(* CODESYS project GitDemo

Project tree, tasks and I/O mapping:
  XC204_1 : XC204, Eaton Automation, version 3.5.19.61
      unmapped channels: Output, Input
    application Application
      libraries: Standard, 3.5.18.0 (System); EA_XN300_CAN, 3.5.19.30 (Eaton Automation); EA_XN322_2SI_RS, 3.5.18.2 (Eaton Automation); EA_XN300local_ext, 3.5.19.30 (Eaton Automation)
      task EtherCAT_Task (cyclic, interval t#4ms, priority 1) calls nothing
      task MainTask (cyclic, interval t#10ms, priority 1) calls PLC_PRG, XN300Local
      program PLC_PRG [ST]
      program XN300Local [ST]
    EtherCAT_Master : EtherCAT Master, CODESYS, version 4.8.0.0
        settings: SlaveAutoRestart = True; NetworkName = 'eth1'; NetworkName = "eth1"; SrcAddress1 = 5; SrcAddress2 = 1258783711
      XN_312_GW_EC_1 : XN-312-GW-EC (Eaton SDIAS XN-312-GW-EtherCAT Gateway), Eaton Industries GmbH, order no. XN-312-GW-EC, version Revision=16#00000000
          settings: StationAlias = 0; DC sync0 cycletime = 4000; DC sync1 cycletime = 4000
    XN300_Master : XN300-Master, Eaton Automation, version 3.5.10.0
      XN_322_20DI_PD : XN-322-20DI-PD, Eaton Automation, order no. 8001, version 3.5.10.0
          unmapped channels: Inputs
      XN_322_2DMS_WM_1 : XN-322-2DMS-WM, Eaton Automation, order no. 8006, version 3.5.10.0
          unmapped channels: InputChannel1, InputChannel2, ADC1Diag, ADC2Diag, ModuleDiag
      XN_322_8AIO_I_1 : XN-322-8AIO-I, Eaton Automation, order no. 8012, version 3.5.20.0
          unmapped channels: OutputChannel1, OutputChannel2, OutputChannel3, OutputChannel4, InputChannel1, InputChannel2, InputChannel3, InputChannel4, ModuleDiag, WireBreakDiag
  XC204 : XC204, Eaton Automation, version 3.5.19.61
      unmapped channels: Output, Input
    application Application
      libraries: EA_XN300_CAN, 3.5.19.30 (Eaton Automation); Standard, 3.5.18.0 (System); CAA CiA 405, 4.1.0.0 (CAA Technical Workgroup); MemoryUtils, * (3S - Smart Software Solutions GmbH); StringUtils, 3.5.18.0 (System)
      task MainTask (cyclic, interval t#10ms, priority 1) calls CANopenEnDisableDeviceExample, CANopenManagerExamples, CANbusExamples
      CANbus Examples/
        program CANbusExamples [ST]
        Change CANbus settings (Reconfigure)/
          program ChangeBaudrate [ST]
          program EnableDisableCANbus [ST]
        Query CANbus/
          function GetCANbus [ST]
      CANopen Master Examples/
        program CANopenManagerExamples [ST]
        CiA405/
          Diagnosis/
            EMCY/
              program ReceiveEMCYFromAllDevicesExample [ST]
              program ReceiveEMCYFromOneDeviceExample [ST]
            State/
              program GetCANopenKernelStateExample [ST]
              program GetStateExample [ST]
          Network management/
            program GetCANopenManagerNodeIDExample [ST]
            program NMT_Example [ST]
          SDO access/
            Block and Segmented/
              program SegmentedAndBlockReadExample [ST]
              program SegmentedAndBlockWriteExample [ST]
            Expedited (<= 4byte)/
              program ExpeditedReadExample [ST]
              program ExpeditedWriteExample [ST]
        Stack API/
          program CANopenManagerAPI [ST]
          program CANopenRemoteDeviceAPI [ST]
          Events/
            function block CANopenManagerEventHandler [ST]: EventCallback
      program CANopenEnDisableDeviceExample [ST]
    CANbus : CANbus, Eaton Automation, version 4.2.0.0
      CANopen_Manager : CANopen_Manager, Eaton Automation, version 4.2.0.0
          settings: ConfigVersion = 50659584
        XN_312_GW_CAN : XN-312-GW-CAN, Eaton Automation, order no. 178782, version Revision=16#00000000, FileVersion=1.12
            settings: NODEIDSAVED = 2; SDO Timeout = 1000000; PDO_Autoconfig = TRUE; EXPERTSETTINGS = True; Nodeguarding.Guard Time = 0 ms; Nodeguarding.Life Time Factor = 0; Emergency-General Parameters.Emergency COBID = 16#00000082; Heartbeat-Producer Time = 200; Settings.COBID = 16#00000202; Settings.Transmission Type = 16#FF; Settings.available PDO-Parameter.Inhibit Time available = FALSE; Settings.available PDO-Parameter.Event Timer available = FALSE; Settings.Inhibit Time = 0; Settings.Event Timer = 0; Generic COBID = '$NODEID+16#0200'; Process by CANopenManager = TRUE; Settings.COBID = 16#00000182; Settings.Transmission Type = 16#FF; Settings.available PDO-Parameter.Inhibit Time available = TRUE; Settings.available PDO-Parameter.Event Timer available = TRUE; Settings.Inhibit Time = 0; Settings.Event Timer = 0; Generic COBID = '$NODEID+16#0180'; Process by CANopenManager = TRUE; Settings.COBID = 16#00000282; Settings.Transmission Type = 16#FF; Settings.available PDO-Parameter.Inhibit Time available = TRUE; Settings.available PDO-Parameter.Event Timer available = TRUE; Settings.Inhibit Time = 0; Settings.Event Timer = 0; Generic COBID = '$NODEID+16#0280'; Process by CANopenManager = TRUE; Heartbeat-Consuming1.Heartbeat-Time = 300 ms; Q-Byte : XN_322_16MIO_DIOAI.Index = 16#6200; Q-Byte : XN_322_16MIO_DIOAI.Subindex = 16#01; Q-Byte : XN_322_16MIO_DIOAI.ObjectLength = 8; I-Byte : XN_322_16MIO_DIOAI.Index = 16#6000; I-Byte : XN_322_16MIO_DIOAI.Subindex = 16#01; I-Byte : XN_322_16MIO_DIOAI.ObjectLength = 8; I-Byte : XN_322_16MIO_DIOAI.Index = 16#6000;
              I-Byte : XN_322_16MIO_DIOAI.Subindex = 16#02; I-Byte : XN_322_16MIO_DIOAI.ObjectLength = 8; I-Byte : XN_322_20DI_PCNT.Index = 16#6000; I-Byte : XN_322_20DI_PCNT.Subindex = 16#03; I-Byte : XN_322_20DI_PCNT.ObjectLength = 8; I-Byte : XN_322_20DI_PCNT.Index = 16#6000; I-Byte : XN_322_20DI_PCNT.Subindex = 16#04; I-Byte : XN_322_20DI_PCNT.ObjectLength = 8; I-Byte : XN_322_20DI_PCNT.Index = 16#6000; I-Byte : XN_322_20DI_PCNT.Subindex = 16#05; I-Byte : XN_322_20DI_PCNT.ObjectLength = 8; I-WORD : XN_322_16MIO_DIOAI.Index = 16#6401; I-WORD : XN_322_16MIO_DIOAI.Subindex = 16#01; I-WORD : XN_322_16MIO_DIOAI.ObjectLength = 16; I-WORD : XN_322_16MIO_DIOAI.Index = 16#6401; I-WORD : XN_322_16MIO_DIOAI.Subindex = 16#02; I-WORD : XN_322_16MIO_DIOAI.ObjectLength = 16; SDO List.Set COB-ID sync.Index = 16#1005; SDO List.Set COB-ID sync.Subindex = 16#00; SDO List.Set COB-ID sync.Value = 16#00000080; SDO List.Set COB-ID sync.Size = 32; SDO List.Set COB-ID sync.AbortIfError = FALSE; SDO List.Set COB-ID sync.JumpToLine = FALSE; SDO List.Set COB-ID sync.Line = 0; SDO List.Set Guardtime.Index = 16#100C; SDO List.Set Guardtime.Subindex = 16#00; SDO List.Set Guardtime.Value = 16#00000000; SDO List.Set Guardtime.Size = 16; SDO List.Set Guardtime.AbortIfError = FALSE; SDO List.Set Guardtime.JumpToLine = FALSE; SDO List.Set Guardtime.Line = 0; SDO List.Set Lifetime.Index = 16#100D; SDO List.Set Lifetime.Subindex = 16#00; SDO List.Set Lifetime.Value = 16#00000000; SDO List.Set Lifetime.Size = 8; SDO List.Set Lifetime.AbortIfError = FALSE; SDO List.Set Lifetime.JumpToLine = FALSE; SDO List.Set Lifetime.Line = 0; SDO List.Disable Emcy CobID.Index = 16#1014; SDO List.Disable Emcy CobID.Subindex = 16#00;
              SDO List.Disable Emcy CobID.Value = 16#80000082; SDO List.Disable Emcy CobID.Size = 32; SDO List.Disable Emcy CobID.AbortIfError = FALSE; SDO List.Disable Emcy CobID.JumpToLine = FALSE; SDO List.Disable Emcy CobID.Line = 0; SDO List.Set Emcy CobID.Index = 16#1014; SDO List.Set Emcy CobID.Subindex = 16#00; SDO List.Set Emcy CobID.Value = 16#00000082; SDO List.Set Emcy CobID.Size = 32; SDO List.Set Emcy CobID.AbortIfError = FALSE; SDO List.Set Emcy CobID.JumpToLine = FALSE; SDO List.Set Emcy CobID.Line = 0; SDO List.Set Heartbeat Consumer.Index = 16#1016; SDO List.Set Heartbeat Consumer.Subindex = 16#01; SDO List.Set Heartbeat Consumer.Value = 16#0001012C; SDO List.Set Heartbeat Consumer.Size = 32; SDO List.Set Heartbeat Consumer.AbortIfError = FALSE; SDO List.Set Heartbeat Consumer.JumpToLine = FALSE; SDO List.Set Heartbeat Consumer.Line = 0; SDO List.Set Heartbeat Consumer.Index = 16#1016; SDO List.Set Heartbeat Consumer.Subindex = 16#02; SDO List.Set Heartbeat Consumer.Value = 0; SDO List.Set Heartbeat Consumer.Size = 32; SDO List.Set Heartbeat Consumer.AbortIfError = FALSE; SDO List.Set Heartbeat Consumer.JumpToLine = FALSE; SDO List.Set Heartbeat Consumer.Line = 0; SDO List.Set Heartbeat Consumer.Index = 16#1016; SDO List.Set Heartbeat Consumer.Subindex = 16#03; SDO List.Set Heartbeat Consumer.Value = 0; SDO List.Set Heartbeat Consumer.Size = 32; SDO List.Set Heartbeat Consumer.AbortIfError = FALSE; SDO List.Set Heartbeat Consumer.JumpToLine = FALSE; SDO List.Set Heartbeat Consumer.Line = 0; SDO List.Set Heartbeat Consumer.Index = 16#1016; SDO List.Set Heartbeat Consumer.Subindex = 16#04; SDO List.Set Heartbeat Consumer.Value = 0; SDO List.Set Heartbeat Consumer.Size = 32; SDO List.Set Heartbeat Consumer.AbortIfError = FALSE; SDO List.Set Heartbeat Consumer.JumpToLine = FALSE; SDO List.Set Heartbeat Consumer.Line = 0;
              SDO List.Set Heartbeat Producer.Index = 16#1017; SDO List.Set Heartbeat Producer.Subindex = 16#00; SDO List.Set Heartbeat Producer.Value = 16#000000C8; SDO List.Set Heartbeat Producer.Size = 16; SDO List.Set Heartbeat Producer.AbortIfError = FALSE; SDO List.Set Heartbeat Producer.JumpToLine = FALSE; SDO List.Set Heartbeat Producer.Line = 0; SDO List.Disable PDO.Index = 16#1400; SDO List.Disable PDO.Subindex = 16#01; SDO List.Disable PDO.Value = 16#80000202; SDO List.Disable PDO.Size = 32; SDO List.Disable PDO.AbortIfError = FALSE; SDO List.Disable PDO.JumpToLine = FALSE; SDO List.Disable PDO.Line = 0; SDO List.Set transmission type.Index = 16#1400; SDO List.Set transmission type.Subindex = 16#02; SDO List.Set transmission type.Value = 16#FF; SDO List.Set transmission type.Size = 8; SDO List.Set transmission type.AbortIfError = FALSE; SDO List.Set transmission type.JumpToLine = FALSE; SDO List.Set transmission type.Line = 0; SDO List.Clear pdo mapping.Index = 16#1600; SDO List.Clear pdo mapping.Subindex = 16#00; SDO List.Clear pdo mapping.Value = 16#0; SDO List.Clear pdo mapping.Size = 8; SDO List.Clear pdo mapping.AbortIfError = FALSE; SDO List.Clear pdo mapping.JumpToLine = FALSE; SDO List.Clear pdo mapping.Line = 0; SDO List.Set Mapping.Index = 16#1600; SDO List.Set Mapping.Subindex = 16#01; SDO List.Set Mapping.Value = 16#62000108; SDO List.Set Mapping.Size = 32; SDO List.Set Mapping.AbortIfError = FALSE; SDO List.Set Mapping.JumpToLine = FALSE; SDO List.Set Mapping.Line = 0; SDO List.Set number of mappings.Index = 16#1600; SDO List.Set number of mappings.Subindex = 16#00; SDO List.Set number of mappings.Value = 16#01; SDO List.Set number of mappings.Size = 8; SDO List.Set number of mappings.AbortIfError = FALSE;
              SDO List.Set number of mappings.JumpToLine = FALSE; SDO List.Set number of mappings.Line = 0; SDO List.Set and enable COB-ID.Index = 16#1400; SDO List.Set and enable COB-ID.Subindex = 16#01; SDO List.Set and enable COB-ID.Value = 16#00000202; SDO List.Set and enable COB-ID.Size = 32; SDO List.Set and enable COB-ID.AbortIfError = FALSE; SDO List.Set and enable COB-ID.JumpToLine = FALSE; SDO List.Set and enable COB-ID.Line = 0; SDO List.Disable PDO.Index = 16#1800; SDO List.Disable PDO.Subindex = 16#01; SDO List.Disable PDO.Value = 16#80000182; SDO List.Disable PDO.Size = 32; SDO List.Disable PDO.AbortIfError = FALSE; SDO List.Disable PDO.JumpToLine = FALSE; SDO List.Disable PDO.Line = 0; SDO List.Set transmission type.Index = 16#1800; SDO List.Set transmission type.Subindex = 16#02; SDO List.Set transmission type.Value = 16#FF; SDO List.Set transmission type.Size = 8; SDO List.Set transmission type.AbortIfError = FALSE; SDO List.Set transmission type.JumpToLine = FALSE; SDO List.Set transmission type.Line = 0; SDO List.Set inhibit time.Index = 16#1800; SDO List.Set inhibit time.Subindex = 16#03; SDO List.Set inhibit time.Value = 16#0000; SDO List.Set inhibit time.Size = 16; SDO List.Set inhibit time.AbortIfError = FALSE; SDO List.Set inhibit time.JumpToLine = FALSE; SDO List.Set inhibit time.Line = 0; SDO List.Set event time.Index = 16#1800; SDO List.Set event time.Subindex = 16#05; SDO List.Set event time.Value = 16#0000; SDO List.Set event time.Size = 16; SDO List.Set event time.AbortIfError = FALSE; SDO List.Set event time.JumpToLine = FALSE; SDO List.Set event time.Line = 0; SDO List.Clear pdo mapping.Index = 16#1A00; SDO List.Clear pdo mapping.Subindex = 16#00; SDO List.Clear pdo mapping.Value = 16#0;
              SDO List.Clear pdo mapping.Size = 8; SDO List.Clear pdo mapping.AbortIfError = FALSE; SDO List.Clear pdo mapping.JumpToLine = FALSE; SDO List.Clear pdo mapping.Line = 0; SDO List.Set Mapping.Index = 16#1A00; SDO List.Set Mapping.Subindex = 16#01; SDO List.Set Mapping.Value = 16#60000108; SDO List.Set Mapping.Size = 32; SDO List.Set Mapping.AbortIfError = FALSE; SDO List.Set Mapping.JumpToLine = FALSE; SDO List.Set Mapping.Line = 0; SDO List.Set Mapping.Index = 16#1A00; SDO List.Set Mapping.Subindex = 16#02; SDO List.Set Mapping.Value = 16#60000208; SDO List.Set Mapping.Size = 32; SDO List.Set Mapping.AbortIfError = FALSE; SDO List.Set Mapping.JumpToLine = FALSE; SDO List.Set Mapping.Line = 0; SDO List.Set Mapping.Index = 16#1A00; SDO List.Set Mapping.Subindex = 16#03; SDO List.Set Mapping.Value = 16#60000308; SDO List.Set Mapping.Size = 32; SDO List.Set Mapping.AbortIfError = FALSE; SDO List.Set Mapping.JumpToLine = FALSE; SDO List.Set Mapping.Line = 0; SDO List.Set Mapping.Index = 16#1A00; SDO List.Set Mapping.Subindex = 16#04; SDO List.Set Mapping.Value = 16#60000408; SDO List.Set Mapping.Size = 32; SDO List.Set Mapping.AbortIfError = FALSE; SDO List.Set Mapping.JumpToLine = FALSE; SDO List.Set Mapping.Line = 0; SDO List.Set Mapping.Index = 16#1A00; SDO List.Set Mapping.Subindex = 16#05; SDO List.Set Mapping.Value = 16#60000508; SDO List.Set Mapping.Size = 32; SDO List.Set Mapping.AbortIfError = FALSE; SDO List.Set Mapping.JumpToLine = FALSE; SDO List.Set Mapping.Line = 0; SDO List.Set number of mappings.Index = 16#1A00;
              SDO List.Set number of mappings.Subindex = 16#00; SDO List.Set number of mappings.Value = 16#05; SDO List.Set number of mappings.Size = 8; SDO List.Set number of mappings.AbortIfError = FALSE; SDO List.Set number of mappings.JumpToLine = FALSE; SDO List.Set number of mappings.Line = 0; SDO List.Set and enable COB-ID.Index = 16#1800; SDO List.Set and enable COB-ID.Subindex = 16#01; SDO List.Set and enable COB-ID.Value = 16#00000182; SDO List.Set and enable COB-ID.Size = 32; SDO List.Set and enable COB-ID.AbortIfError = FALSE; SDO List.Set and enable COB-ID.JumpToLine = FALSE; SDO List.Set and enable COB-ID.Line = 0; SDO List.Disable PDO.Index = 16#1801; SDO List.Disable PDO.Subindex = 16#01; SDO List.Disable PDO.Value = 16#80000282; SDO List.Disable PDO.Size = 32; SDO List.Disable PDO.AbortIfError = FALSE; SDO List.Disable PDO.JumpToLine = FALSE; SDO List.Disable PDO.Line = 0; SDO List.Set transmission type.Index = 16#1801; SDO List.Set transmission type.Subindex = 16#02; SDO List.Set transmission type.Value = 16#FF; SDO List.Set transmission type.Size = 8; SDO List.Set transmission type.AbortIfError = FALSE; SDO List.Set transmission type.JumpToLine = FALSE; SDO List.Set transmission type.Line = 0; SDO List.Set inhibit time.Index = 16#1801; SDO List.Set inhibit time.Subindex = 16#03; SDO List.Set inhibit time.Value = 16#0000; SDO List.Set inhibit time.Size = 16; SDO List.Set inhibit time.AbortIfError = FALSE; SDO List.Set inhibit time.JumpToLine = FALSE; SDO List.Set inhibit time.Line = 0; SDO List.Set event time.Index = 16#1801; SDO List.Set event time.Subindex = 16#05; SDO List.Set event time.Value = 16#0000; SDO List.Set event time.Size = 16; SDO List.Set event time.AbortIfError = FALSE; SDO List.Set event time.JumpToLine = FALSE;
              SDO List.Set event time.Line = 0; SDO List.Clear pdo mapping.Index = 16#1A01; SDO List.Clear pdo mapping.Subindex = 16#00; SDO List.Clear pdo mapping.Value = 16#0; SDO List.Clear pdo mapping.Size = 8; SDO List.Clear pdo mapping.AbortIfError = FALSE; SDO List.Clear pdo mapping.JumpToLine = FALSE; SDO List.Clear pdo mapping.Line = 0; SDO List.Set Mapping.Index = 16#1A01; SDO List.Set Mapping.Subindex = 16#01; SDO List.Set Mapping.Value = 16#64010110; SDO List.Set Mapping.Size = 32; SDO List.Set Mapping.AbortIfError = FALSE; SDO List.Set Mapping.JumpToLine = FALSE; SDO List.Set Mapping.Line = 0; SDO List.Set Mapping.Index = 16#1A01; SDO List.Set Mapping.Subindex = 16#02; SDO List.Set Mapping.Value = 16#64010210; SDO List.Set Mapping.Size = 32; SDO List.Set Mapping.AbortIfError = FALSE; SDO List.Set Mapping.JumpToLine = FALSE; SDO List.Set Mapping.Line = 0; SDO List.Set number of mappings.Index = 16#1A01; SDO List.Set number of mappings.Subindex = 16#00; SDO List.Set number of mappings.Value = 16#02; SDO List.Set number of mappings.Size = 8; SDO List.Set number of mappings.AbortIfError = FALSE; SDO List.Set number of mappings.JumpToLine = FALSE; SDO List.Set number of mappings.Line = 0; SDO List.Set and enable COB-ID.Index = 16#1801; SDO List.Set and enable COB-ID.Subindex = 16#01; SDO List.Set and enable COB-ID.Value = 16#00000282; SDO List.Set and enable COB-ID.Size = 32; SDO List.Set and enable COB-ID.AbortIfError = FALSE; SDO List.Set and enable COB-ID.JumpToLine = FALSE; SDO List.Set and enable COB-ID.Line = 0; ConfigVersion = 50659584
          XN_322_16MIO_DIOAI : XN-322-16MIO-DIOAI, Eaton Automation, order no. 0, version Revision=16#00000000, FileVersion=1.12
              settings: Number of Params = 1; Q-Byte : XN_322_16MIO_DIOAI.Index = 16#6200; Q-Byte : XN_322_16MIO_DIOAI.Subindex = 16#01; Q-Byte : XN_322_16MIO_DIOAI.Startbit = 0; Q-Byte : XN_322_16MIO_DIOAI.Endbit = 7; Number of Params = 4; I-Byte : XN_322_16MIO_DIOAI.Index = 16#6000; I-Byte : XN_322_16MIO_DIOAI.Subindex = 16#01; I-Byte : XN_322_16MIO_DIOAI.Startbit = 0; I-Byte : XN_322_16MIO_DIOAI.Endbit = 7; I-Byte : XN_322_16MIO_DIOAI.Index = 16#6000; I-Byte : XN_322_16MIO_DIOAI.Subindex = 16#02; I-Byte : XN_322_16MIO_DIOAI.Startbit = 0; I-Byte : XN_322_16MIO_DIOAI.Endbit = 7; I-WORD : XN_322_16MIO_DIOAI.Index = 16#6401; I-WORD : XN_322_16MIO_DIOAI.Subindex = 16#01; I-WORD : XN_322_16MIO_DIOAI.Startbit = 0; I-WORD : XN_322_16MIO_DIOAI.Endbit = 15; I-WORD : XN_322_16MIO_DIOAI.Index = 16#6401; I-WORD : XN_322_16MIO_DIOAI.Subindex = 16#02; I-WORD : XN_322_16MIO_DIOAI.Startbit = 0; I-WORD : XN_322_16MIO_DIOAI.Endbit = 15
              unmapped channels: Q-Byte : XN_322_16MIO_DIOAI, I-Byte : XN_322_16MIO_DIOAI, I-Byte : XN_322_16MIO_DIOAI, I-WORD : XN_322_16MIO_DIOAI, I-WORD : XN_322_16MIO_DIOAI
          XN_322_20DI_PCNT : XN-322-20DI-PCNT, Eaton Automation, order no. 0, version Revision=16#00000000, FileVersion=1.12
              settings: Number of Params = 3; I-Byte : XN_322_20DI_PCNT.Index = 16#6000; I-Byte : XN_322_20DI_PCNT.Subindex = 16#03; I-Byte : XN_322_20DI_PCNT.Startbit = 0; I-Byte : XN_322_20DI_PCNT.Endbit = 7; I-Byte : XN_322_20DI_PCNT.Index = 16#6000; I-Byte : XN_322_20DI_PCNT.Subindex = 16#04; I-Byte : XN_322_20DI_PCNT.Startbit = 0; I-Byte : XN_322_20DI_PCNT.Endbit = 7; I-Byte : XN_322_20DI_PCNT.Index = 16#6000; I-Byte : XN_322_20DI_PCNT.Subindex = 16#05; I-Byte : XN_322_20DI_PCNT.Startbit = 0; I-Byte : XN_322_20DI_PCNT.Endbit = 7
              unmapped channels: I-Byte : XN_322_20DI_PCNT, I-Byte : XN_322_20DI_PCNT, I-Byte : XN_322_20DI_PCNT
          XN_322_2SI_RS : XN-322-2SI-RS, Eaton Automation, order no. 0, version Revision=16#00000000, FileVersion=1.12
  text list GlobalTextList
*)

// XC204_1/Application/PLC_PRG
PROGRAM PLC_PRG
VAR
    iState 		: INT := 0;
    reconfig 	: DED.Reconfigure;
	xDisable	: BOOL;
	xEnable	: BOOL;
	fbTRIG_Disable: R_TRIG;
	fbTRIG_Enable: R_TRIG;
	xError: BOOL;
	xDone: BOOL;
END_VAR

fbTRIG_Disable(CLK:= xDisable, Q=> );
fbTRIG_Enable(CLK:= xEnable , Q=> );

(*
CASE iState OF
	
	0: //Enable/Disable slave device: Slave1 (= name in device tree) 
		IF fbTRIG_Enable.Q THEN
			XN_312_GW_CAN.Enable := TRUE;
			XN300_Master.Enable := TRUE;
			xError := FALSE;
			iState := 1;
		ELSIF fbTRIG_Disable.Q THEN
			XN_312_GW_CAN.Enable := FALSE;
			XN300_Master.Enable := FALSE;
			xError := FALSE;
			iState := 1;
		END_IF

    1: //start reconfiguring of fieldbus master
      reconfig(xExecute := TRUE, itfNode := CANopen_Manager);
       IF reconfig.xDone THEN
           iState := 3;
       ELSIF reconfig.xError THEN
           iState := 2;
       END_IF

    2: //reconfiguring error
       //TODO: Add code here
       reconfig(xExecute := FALSE);	
	   xError := TRUE;
	   iState := 0;

    3: //reconfiguring successful ==> slave disabled
       //TODO: Add code here
       reconfig(xExecute := FALSE);
	   xDone := TRUE;
	   iState := 0;

END_CASE

*)

END_PROGRAM

// XC204_1/Application/XN300Local
PROGRAM XN300Local
VAR
	eMasterStatusInfo1: ENUM_MASTERSTATUSINFO;
	sMasterStatusInfo2: STRING;
	uiPeriode: UINT;
	stSlotInfo: EA_XN300local_ext.STRUCT_XNSLOTINFO;
	byData: BYTE;
	xRead: BOOL;
END_VAR

// Get XN300_Master Status
GetXnMasterStatus(peStatusInfo:= ADR(eMasterStatusInfo1), pstrStatusInfo2:= ADR(sMasterStatusInfo2), uiStatusInfo2Length:= LEN(sMasterStatusInfo2));

uiPeriode := GetXnPeriode();

stSlotInfo := GetXnSlotInfo(uiSlotNumber:= 1);

// XN_322_8AO_U2 -> Offset 16#80 -> ModuleDiagnose 1:No power supply, 2:No SyncSignal, 3: FlashCRC Error, 4:RAMCRC Error, 5:FlashMemory Error
IF xRead THEN
	ReadXnDirect(uiModuleNumber:= 1, uiModuleOffset:=16#080 , uiDataLength:= 2, pbyData:= ADR(byData));
	xRead := FALSE;
END_IF

(*
SetXnPeriode(uiXnPeriode:= );

SetXnUserLed(uiModuleNumber:= , uiLedMode:= );

WriteXnDirect(uiModuleNumber:= , uiModuleOffset:= , uiDataLength:= , pbyData:= );
*)

END_PROGRAM

// XC204/Application/CANopenEnDisableDeviceExample
PROGRAM CANopenEnDisableDeviceExample
VAR
    iState 		: INT := 0;
    reconfig 	: DED.Reconfigure;
	xDisable	: BOOL;
	xEnable	: BOOL;
	fbTRIG_Disable: R_TRIG;
	fbTRIG_Enable: R_TRIG;
	xError: BOOL;
	xDone: BOOL;
END_VAR

fbTRIG_Disable(CLK:= xDisable, Q=> );
fbTRIG_Enable(CLK:= xEnable , Q=> );


CASE iState OF
	
	0: //Enable/Disable slave device: Slave1 (= name in device tree) 
		IF fbTRIG_Enable.Q THEN
			XN_312_GW_CAN.Enable := TRUE;
			xError := FALSE;
			iState := 1;
		ELSIF fbTRIG_Disable.Q THEN
			XN_312_GW_CAN.Enable := FALSE;
			xError := FALSE;
			iState := 1;
		END_IF

    1: //start reconfiguring of fieldbus master
      reconfig(xExecute := TRUE, itfNode := CANopen_Manager);
       IF reconfig.xDone THEN
           	iState := 3;
			xDisable := FALSE;
			xEnable := FALSE;
       ELSIF reconfig.xError THEN
           iState := 2;
       END_IF

    2: //reconfiguring error
       //TODO: Add code here
       reconfig(xExecute := FALSE);	
	   xError := TRUE;
	   iState := 0;

    3: //reconfiguring successful ==> slave disabled
       //TODO: Add code here
       reconfig(xExecute := FALSE);
	   xDone := TRUE;
	   iState := 0;

END_CASE

END_PROGRAM

// XC204/Application/CANopen Master Examples/CANopenManagerExamples
PROGRAM CANopenManagerExamples
VAR
END_VAR

///////////////////////////////////////// CIA 405 Examples //////////////////////////////////////////////////////

//Diagnosis Examples
GetStateExample(); //How to get the state of a CANopenRemote Device?
GetCANopenKernelStateExample(); //How to get the CANopen stack kernel state?
ReceiveEMCYFromAllDevicesExample(); //How to check if any CANopenRemote Device has a pending Emergency?
ReceiveEMCYFromOneDeviceExample(); //How to check if a specific CANopenRemote Device has a pending Emergency?

//SDO Examples
ExpeditedReadExample(); //How to read up to 4 bytes by SDO?
ExpeditedWriteExample(); //How to write up to 4 bytes by SDO?
SegmentedAndBlockReadExample(); //How to read more than 4 bytes by SDO?
SegmentedAndBlockWriteExample(); //How to write more than 4 bytes by SDO?

NMT_Example(); //How to start/stop/reset CANopenRemote Devices?

GetCANopenManagerNodeIDExample(); //How to read the CANopen Manager NodeID?

///////////////////////////////////////// General Examples //////////////////////////////////////////////////////

CANopenManagerAPI(); //How to use the CANopen Manager API?
CANopenRemoteDeviceAPI(); //How to use the CANopenRemoteDevice API?

END_PROGRAM

// XC204/Application/CANopen Master Examples/CiA405/Diagnosis/State/GetStateExample
// The following program gets the current CANopen state of the CANopenRemoteDevice attached below the CANopen_Manager.
// Set xEnable to TRUE in online mode to get the program working.
PROGRAM GetStateExample
VAR
	xEnable : BOOL; // Set this variable to true to start the example code. Variable will be set to FALSE if GetState finished execution.
	State : CiA405.DEVICE_STATE; // Result: CANopen State
	
	GetState : CIA405.GET_STATE;
END_VAR

IF GetState.CONFIRM = TRUE THEN
	// GetState successful. Output STATE contains result.
	State := GetState.STATE;
	xEnable := FALSE;
ELSIF GetState.ERROR <> CIA405.CANOPEN_KERNEL_ERROR.CANOPEN_KERNEL_NO_ERROR THEN
	// an error occured while processing GetState e.g. wrong NodeID or NetworkID
	xEnable := FALSE;
END_IF

// GetState needs the CAN network and the device NodeID (input DEVICE). 
GetState( 	ENABLE := xEnable,
		  	NETWORK := CANbus.NetId + 1, //CODESYS NetId starts by 0 (the number entered into the CANbus configurator); CiA405 NETWORK by 1; That is the reason why we have to increment it here.
		  	TIMEOUT := 0, // no timeout for GetState needed because it is processed locally.
			DEVICE := XN_312_GW_CAN.NodeID // Note: If you want to get the state of the CANopenManager, you can use the CANopenManager NodeID or NodeID 0.
												 // A CANopenManager goes to OPERATIONAL if all mandatory (= not optional) slaves are operational.
);

END_PROGRAM

// XC204/Application/CANopen Master Examples/CiA405/Diagnosis/State/GetCANopenKernelStateExample
// This program gets the state of the CANopenManager kernel. If kernel has no error everything is working fine.
// See CiA405.CANOPEN_KERNEL_ERROR in library manager for further details.
// Set xEnable to TRUE in online mode to get the program working.
PROGRAM GetCANopenKernelStateExample
VAR
	xEnable : BOOL; // Set this variable to true to start the example code. Variable will be set to FALSE if GetState finished execution.
	xErrorPending : BOOL; //true if a CANopen Kernel error is pending
	State : CiA405.CANOPEN_KERNEL_ERROR; // Result: CANopen Manager kernel state
	
	GetKernelState : CIA405.GET_CANOPEN_KERNEL_STATE;
END_VAR

IF GetKernelState.CONFIRM = TRUE THEN
	// GetKernelState successful. Output STATE contains result.
	State := GetKernelState.STATE;
	xErrorPending := State <> CIA405.CANOPEN_KERNEL_ERROR.CANOPEN_KERNEL_NO_ERROR;
	xEnable := FALSE;
ELSIF GetKernelState.ERROR <> CIA405.CANOPEN_KERNEL_ERROR.CANOPEN_KERNEL_NO_ERROR THEN
	// an error occured while processing GetKernelState e.g. wrong NetworkID
	xEnable := FALSE;
END_IF

GetKernelState( 	ENABLE := xEnable,
		  			NETWORK := CANbus.NetId + 1, //CODESYS NetId starts by 0 (the number entered into the CANbus configurator); CiA405 NETWORK by 1; That is the reason why we have to increment it here.
		  			TIMEOUT := 0 // no timeout for GetKernelState needed because it is processed locally.
);

END_PROGRAM

// XC204/Application/CANopen Master Examples/CiA405/Diagnosis/EMCY/ReceiveEMCYFromAllDevicesExample
// This program checks if any emergency is pending for any device of a given CANopenManager network.
// Set xEnable to TRUE in online mode to get the program working.
PROGRAM ReceiveEMCYFromAllDevicesExample
VAR
	xEnable : BOOL; // Set this variable to true to start the example code. Variable will be set to FALSE if RecvEMCY finished execution.
	xEMCYPending : BOOL; //true if EMCY is pending ==> see EMCY and NodeID for EMCY information
	EMCY : CIA405.EMCY_ERROR; //contains EMCY information
	NodeID : CIA405.DEVICE; //NodeID of EMCY sender
	
	RecvEMCY : CIA405.RECV_EMCY;
END_VAR

IF RecvEMCY.CONFIRM = TRUE THEN
	// RecvEMCY successful.
	IF RecvEMCY.DEVICE <> 0 THEN
		//an EMCY from NodeID RecvEMCY.DEVICE is pending
		xEMCYPending := TRUE;
		EMCY := RecvEMCY.ERRORINFO;
		NodeID := RecvEMCY.DEVICE;
	ELSE
		//all devices are error free
		xEMCYPending := FALSE;
	END_IF

	xEnable := FALSE;
ELSIF RecvEMCY.ERROR <> CIA405.CANOPEN_KERNEL_ERROR.CANOPEN_KERNEL_NO_ERROR THEN
	// an error occured while processing RecvEMCY e.g. wrong NodeID or NetworkID
	xEnable := FALSE;
END_IF

RecvEMCY( 	ENABLE := xEnable,
		  	NETWORK := CANbus.NetId + 1, //CODESYS NetId starts by 0 (the number entered into the CANbus configurator); CiA405 NETWORK by 1; That is the reason why we have to increment it here.
		  	TIMEOUT := 0 // no timeout for RecvEMCY needed because it is processed locally.
);

END_PROGRAM

// XC204/Application/CANopen Master Examples/CiA405/Diagnosis/EMCY/ReceiveEMCYFromOneDeviceExample
// This program checks if any emergency is pending for CANopenRemoteDevice.
// Set xEnable to TRUE in online mode to get the program working.
PROGRAM ReceiveEMCYFromOneDeviceExample
VAR
	xEnable : BOOL; // Set this variable to true to start the example code. Variable will be set to FALSE if RecvEMCYDev finished execution.
	xEMCYPending : BOOL; //true if EMCY is pending ==> see EMCY for EMCY information
	EMCY : CIA405.EMCY_ERROR; //contains EMCY information
	
	RecvEMCYDev : CIA405.RECV_EMCY_DEV;
END_VAR

IF RecvEMCYDev.CONFIRM = TRUE THEN
	// RecvEMCYDev successful
	IF RecvEMCYDev.ERRORINFO.EMCY_ERROR_CODE <> 0 THEN
		//an EMCY is pending ==> see RecvEMCYDev.ERRORINFO for EMCY information
		xEMCYPending := TRUE;
		EMCY := RecvEMCYDev.ERRORINFO;
	ELSE
		//device is error free
		xEMCYPending := FALSE;
	END_IF
	xEnable := FALSE;
ELSIF RecvEMCYDev.ERROR <> CIA405.CANOPEN_KERNEL_ERROR.CANOPEN_KERNEL_NO_ERROR THEN
	// an error occured while processing RecvEMCY e.g. wrong NodeID or NetworkID
	xEnable := FALSE;
END_IF

RecvEMCYDev( 	ENABLE := xEnable,
		  		NETWORK := CANbus.NetId + 1, //CODESYS NetId starts by 0 (the number entered into the CANbus configurator); CiA405 NETWORK by 1; That is the reason why we have to increment it here.
		  		TIMEOUT := 0, // no timeout for RecvEMCYDev needed because it is processed locally.
				DEVICE := XN_312_GW_CAN.NodeID //NodeID to receive EMCY from
);

END_PROGRAM

// XC204/Application/CANopen Master Examples/CiA405/SDO access/Expedited (<= 4byte)/ExpeditedReadExample
// The following program reads the device type of CANopenRemoteDevice and shows how to usde SDORead4 function block.
// Set xEnable to TRUE in online mode to get the program working.
PROGRAM ExpeditedReadExample
VAR
	xEnable       : BOOL; // Set this variable to true to start the example code. Variable will be set to FALSE if Expedited transfer finished execution.
	dwValue : DWORD; //read value
	dwAbortCode : DWORD; //contains abort code in case of error
	
	SDORead4 	  : CIA405.SDO_READ4;
END_VAR

IF SDORead4.CONFIRM THEN
	//value was read without error
	// ==> Copy data from SDO read function block
	MEMUtils.MemCpy(pbyDest := ADR(dwValue), pbySrc := ADR(SDORead4.DATA[1]), dwSize := SIZEOF(dwValue));
	//==> On big endian systems: dwValue has to be swapped to CANopen byte order (= Little Endian).
	MEMUtils.SwapLocalToIntel(pAddress := ADR(dwValue), iSize := TO_INT(SIZEOF(dwValue))); //function only swaps on big endian systems
	xEnable := FALSE;
ELSIF SDORead4.ERROR <> CiA405.CANOPEN_KERNEL_ERROR.CANOPEN_KERNEL_NO_ERROR THEN
	//Error occured
	IF SDORead4.ERROR = CIA405.CANOPEN_KERNEL_ERROR.CANOPEN_KERNEL_OTHER_ERROR THEN
		//output error info contains abort code in little endian format
		MEMUtils.MemCpy(pbyDest := ADR(dwAbortCode), pbySrc := ADR(SDORead4.ERRORINFO), dwSize := SIZEOF(dwAbortCode));
		MEMUtils.SwapLocalToIntel(pAddress := ADR(dwAbortCode), iSize := TO_INT(SIZEOF(dwAbortCode))); //function only swaps on big endian systems	
	END_IF
	xEnable := FALSE;
END_IF

SDORead4(
	NETWORK:= CANbus.NetId + 1, //CODESYS NetId starts by 0 (the number entered into the CANbus configurator); CiA405 NETWORK by 1; That is the reason why we have to increment it here.
	ENABLE:= xEnable,
	TIMEOUT:= 0, //Timeout for SDO read in ms. Here: 0 ==> no timeout
	DEVICE:= XN_312_GW_CAN.NodeID, // NodeID of destination device
	CHANNEL:= 0, //SDO channel which should be used. 0 means auto channeling ==> the next free channel will be used. It depends on the slave which settings are working here but 0 and channel 1 is always working. 
	INDEX:= 16#1000, //object index which should be read
	SUBINDEX:= 0 //object sub index which should be read
);

END_PROGRAM

// XC204/Application/CANopen Master Examples/CiA405/SDO access/Expedited (<= 4byte)/ExpeditedWriteExample
// The following program writes a 32bit value with SDO expedited transfer.
// Set xEnable to TRUE in online mode to get the program working.
PROGRAM ExpeditedWriteExample
VAR
	xEnable       : BOOL; // Set this variable to true to start the example code. Variable will be set to FALSE if Expedited transfer finished execution.
	diValue : DINT := 10; //value which should be written
	dwAbortCode : DWORD; //contains abort code in case of error
	
	SDOWrite4 	  : CiA405.SDO_WRITE4;
	RTrig 		  : Standard.R_TRIG;
END_VAR

RTrig(CLK := xEnable); //detect a rising edge for xEnable

IF RTrig.Q THEN
	// Rising edge for xEnable detected ==> Prepare SDO write function block
	// ==> Copy data to SDO write function block
	MEMUtils.MemCpy(pbyDest := ADR(SDOWrite4.DATA[1]), pbySrc := ADR(diValue), dwSize := SIZEOF(diValue));
	//==> On big endian systems: diValue has to be swapped to CANopen byte order (= Little Endian).
	MEMUtils.SwapLocalToIntel(pAddress := ADR(SDOWrite4.DATA[1]), iSize := TO_INT(SIZEOF(diValue))); //function only swaps on big endian systems
END_IF

IF SDOWrite4.CONFIRM THEN
	//value was written without error
	xEnable := FALSE;
ELSIF SDOWrite4.ERROR <> CiA405.CANOPEN_KERNEL_ERROR.CANOPEN_KERNEL_NO_ERROR THEN
	//Error occured
	IF SDOWrite4.ERROR = CIA405.CANOPEN_KERNEL_ERROR.CANOPEN_KERNEL_OTHER_ERROR THEN
		//output error info contains abort code in little endian format
		MEMUtils.MemCpy(pbyDest := ADR(dwAbortCode), pbySrc := ADR(SDOWrite4.ERRORINFO), dwSize := SIZEOF(dwAbortCode));
		MEMUtils.SwapLocalToIntel(pAddress := ADR(dwAbortCode), iSize := TO_INT(SIZEOF(dwAbortCode))); //function only swaps on big endian systems	
	END_IF
	xEnable := FALSE;
END_IF

SDOWrite4(
	NETWORK:= CANbus.NetId + 1, //CODESYS NetId starts by 0 (the number entered into the CANbus configurator); CiA405 NETWORK by 1; That is the reason why we have to increment it here.
	ENABLE:= xEnable,
	TIMEOUT:= 0, //Timeout for SDO write in ms. Here: 0 ==> no timeout
	DEVICE:= XN_312_GW_CAN.NodeID, // NodeID of destination device
	CHANNEL:= 0, //SDO channel which should be used. 0 means auto channeling ==> the next free channel will be used. It depends on the slave which settings are working here but 0 and channel 1 is always working. 
	INDEX:= 16#6412, //object index which should be written
	SUBINDEX:= 1, //object sub index which should be written
	DATALENGTH:= TO_USINT(SIZEOF(diValue)) //length of data to be written
);

END_PROGRAM

// XC204/Application/CANopen Master Examples/CiA405/SDO access/Block and Segmented/SegmentedAndBlockReadExample
// This program uses CiA405.SDO_READ_DATA for reading more than 4 byte from a slave using segmented or block transfer.
//
// This example code reads object 16#1008sub0 which is the device name.
// CiA405.SDO_READ_DATA is a universal function block which can be also used for expedited transfer (<= 4byte).
// If you never want to read more than 4 byte use the CIA405.SDO_READ4 functionblock instead.
// Set xEnable to TRUE in online mode to get the program working.
PROGRAM SegmentedAndBlockReadExample
VAR
	xEnable       : BOOL; // Set this variable to true to start the example code.
	psData        : POINTER TO STRING(MAX_CHAR - 1) := ADR(aData); // Result: Device Name
	dwAbortCode	  : DWORD; //contains abort code in case of error

	SDORead    	  : CIA405.SDO_READ_DATA;
	RTrig 		  : Standard.R_TRIG;										  
	aData	      : ARRAY[0..MAX_CHAR] OF BYTE;
	udiDataLength : UDINT;
END_VAR
VAR CONSTANT
	MAX_CHAR : INT := 256;
END_VAR

RTrig(CLK := xEnable);

IF RTrig.Q THEN
	// Rising edge for xEnable detected ==> Prepare SDO write function block
	
	// ==> Initialize read buffer with 0 (clear old read results)
	MEMUtils.MemSet(pbyBuffer := ADR(aData[0]), byValue := 0, dwSize := SIZEOF(aData));
	
	// ==> Set udiDataLength to read buffer length.
	// Note: Do not forget setting udiDataLength each time when you start a new SDO read operation. 
	// This is necessary because udiDataLength is a VAR_IN_OUT variable and will be modified by SDORead function block!
	// It contains the number of valid bytes read by the function block.
	udiDataLength := SIZEOF(aData) - 1; //-1 only needed because CANopen strings are not null terminated! So we need one additional byte for the null termination. ==> Not needed for other datatypes!
END_IF

IF SDORead.CONFIRM THEN
	// SDO Read successful. aData contains data (= Device Name); udiDataLength contains number of bytes read (string length without null termination).
	xEnable := FALSE;
ELSIF SDORead.ERROR <> CiA405.CANOPEN_KERNEL_ERROR.CANOPEN_KERNEL_NO_ERROR THEN
	// Error occured
	IF SDORead.ERROR = CIA405.CANOPEN_KERNEL_ERROR.CANOPEN_KERNEL_OTHER_ERROR THEN
		//output error info contains abort code in little endian format
		MEMUtils.MemCpy(pbyDest := ADR(dwAbortCode), pbySrc := ADR(SDORead.ERRORINFO), dwSize := SIZEOF(dwAbortCode));
		MEMUtils.SwapLocalToIntel(pAddress := ADR(dwAbortCode), iSize := TO_INT(SIZEOF(dwAbortCode))); //function only swaps on big endian systems	
	END_IF
	xEnable := FALSE;
END_IF

SDORead(   Enable     := xEnable,
		   Network    := CANbus.NetId + 1, //CODESYS NetId starts by 0 (the number entered into the CANbus configurator); CiA405 NETWORK by 1; That is the reason why we have to increment it here.
           Timeout    := 0, //Timeout for SDO read in ms. Here: 0 ==> no timeout
           Device     := XN_312_GW_CAN.NodeID, // NodeID of destination device
           Channel    := 0, //SDO channel which should be used. 0 means auto channeling ==> the next free channel will be used. It depends on the slave which settings are working here but 0 and channel 1 is always working. 
           Index      := 16#1008, //object index which should be read ==> 16#1008sub0 = Device Name
           SubIndex   := 0, //object sub index which should be read ==> 16#1008sub0 = Device Name
		   MODE		  := CIA405.SDO_MODE.AUTO, //Use SDO mode AUTO ==> Mode will be selected automatically. Use SDO_MODE.BLOCK for forcing Block Transfer.
           Data       := ADR(aData), // Pointer to data buffer where result should be written to.
           DataLength := udiDataLength //VAR_IN: Length of data buffer; VAR_OUT: Length of data written to data buffer.
);

END_PROGRAM

// XC204/Application/CANopen Master Examples/CiA405/SDO access/Block and Segmented/SegmentedAndBlockWriteExample
// This program uses CiA405.SDO_WRITE_DATA for writing more than 4 byte using segmented or block transfer.
//
// This example code writes a string into object 16#3000 of CANopenRemoteDevice.
// CiA405.SDO_WRITE_DATA is a universal function block which can be also used for expedited transfer (<= 4byte).
// If you never want to write more than 4 byte use the CIA405.SDO_WRITE4 functionblock instead.
// In online mode: Set psData to the string which should be written and then set xEnable to TRUE to get the program working.
// Afterwards you can check result in CANopenLocalDeviceExamples.strTestString. The Variable is mapped to object 16#3000 in object dictionary.
PROGRAM SegmentedAndBlockWriteExample
VAR
	xEnable       : BOOL; // Set this variable to true to start the example code.
	psData        : POINTER TO STRING(MAX_CHAR - 1) := ADR(aData); // String to write
	dwAbortCode	  : DWORD; //contains abort code in case of error

	SDOWrite      : CIA405.SDO_WRITE_DATA;							  
	aData	      : ARRAY[0..MAX_CHAR] OF BYTE;
END_VAR
VAR CONSTANT
	MAX_CHAR : INT := 256;
END_VAR

IF SDOWrite.CONFIRM THEN
	// SDO Write successful.
	xEnable := FALSE;
ELSIF SDOWrite.ERROR <> CiA405.CANOPEN_KERNEL_ERROR.CANOPEN_KERNEL_NO_ERROR THEN
	// Error occured
	IF SDOWrite.ERROR = CIA405.CANOPEN_KERNEL_ERROR.CANOPEN_KERNEL_OTHER_ERROR THEN
		//output error info contains abort code in little endian format
		MEMUtils.MemCpy(pbyDest := ADR(dwAbortCode), pbySrc := ADR(SDOWrite.ERRORINFO), dwSize := SIZEOF(dwAbortCode));
		MEMUtils.SwapLocalToIntel(pAddress := ADR(dwAbortCode), iSize := TO_INT(SIZEOF(dwAbortCode))); //function only swaps on big endian systems	
	END_IF
	xEnable := FALSE;
END_IF

SDOWrite(  Enable     := xEnable,
		   Network    := CANbus.NetId + 1, //CODESYS NetId starts by 0 (the number entered into the CANbus configurator); CiA405 NETWORK by 1; That is the reason why we have to increment it here.
           Timeout    := 0, //Timeout for SDO read in ms. Here: 0 ==> no timeout
           Device     := XN_312_GW_CAN.NodeID, // NodeID of destination device
           Channel    := 0, //SDO channel which should be used. 0 means auto channeling ==> the next free channel will be used. It depends on the slave which settings are working here but 0 and channel 1 is always working. 
           Index      := 16#3000, //object index which should be written ==> 16#3000 = simple string object
           SubIndex   := 0, //object sub index which should be written
		   MODE		  := CIA405.SDO_MODE.AUTO, //Use SDO mode AUTO ==> Mode will be selected automatically. Use SDO_MODE.BLOCK for forcing Block Transfer.
           Data       := ADR(aData), // Pointer to data buffer where result should be written to.
           DataLength := TO_UDINT(Stu.StrLenA(ADR(aData[0]))) //Length of data
);

END_PROGRAM

// XC204/Application/CANopen Master Examples/CiA405/Network management/NMT_Example
// The following program sends a NMT command to the CANopenRemoteDevice attached below the CANopen_Manager.
// Set eState to the desired NMT command and xEnable to TRUE in online mode to get the program working.
PROGRAM NMT_Example
VAR
	xEnable : BOOL; // Set this variable to true to start the example code. Variable will be set to FALSE if NMT finished execution.
	eState : CIA405.TRANSITION_STATE := CIA405.TRANSITION_STATE.RESET_NODE; // NMT command which should be sent.
	
	NMT : CIA405.NMT;
END_VAR

IF NMT.CONFIRM = TRUE THEN
	// NMT command successful.
	xEnable := FALSE;
ELSIF NMT.ERROR <> CIA405.CANOPEN_KERNEL_ERROR.CANOPEN_KERNEL_NO_ERROR THEN
	// an error occured while processing NMT e.g. wrong NodeID or NetworkID
	xEnable := FALSE;
END_IF

NMT(	ENABLE := xEnable,
		NETWORK := CANbus.NetId + 1, //CODESYS NetId starts by 0 (the number entered into the CANbus configurator); CiA405 NETWORK by 1; That is the reason why we have to increment it here.
		TIMEOUT := 0, // no timeout for GetState needed because it is processed locally.
		DEVICE := XN_312_GW_CAN.NodeID, // Use 0 if you want to send a NMT all command!
		STATE := eState //the NMT command which should be sent
);

END_PROGRAM

// XC204/Application/CANopen Master Examples/CiA405/Network management/GetCANopenManagerNodeIDExample
// This program reads the NodeID of the local CANopenManager.
// Set xEnable to TRUE in online mode to get the program working.
PROGRAM GetCANopenManagerNodeIDExample
VAR
	xEnable : BOOL; // Set this variable to true to start the example code. Variable will be set to FALSE if GetNodeID finished execution.
	NodeID : CiA405.DEVICE; // Result: CANopen NodeID
	
	GetNodeID : CIA405.GET_LOCAL_NODE_ID;
END_VAR

IF GetNodeID.CONFIRM = TRUE THEN
	// GetNodeID successful. Output device contains CANopenManager NodeID.
	NodeID := GetNodeID.DEVICE;
	xEnable := FALSE;
ELSIF GetNodeID.ERROR <> CIA405.CANOPEN_KERNEL_ERROR.CANOPEN_KERNEL_NO_ERROR THEN
	// an error occured while processing GetState e.g. wrong NodeID or NetworkID
	xEnable := FALSE;
END_IF

GetNodeID( 	ENABLE := xEnable,
		  	NETWORK := CANbus.NetId + 1, //CODESYS NetId starts by 0 (the number entered into the CANbus configurator); CiA405 NETWORK by 1; That is the reason why we have to increment it here.
		  	TIMEOUT := 0 // no timeout for GetNodeID needed because it is processed locally.
);

END_PROGRAM

// XC204/Application/CANopen Master Examples/Stack API/CANopenManagerAPI
// This example program shows how to use the CANopen Manager API.
PROGRAM CANopenManagerAPI
VAR
	pDevice : POINTER TO _3SCOS.CANRemoteDevice;
	kernelState : _3SCOS.CANOPEN_KERNEL_STATE;
	xAllMandatorySlaveBooted : BOOL;
	xAllOptionalSlavesBooted : BOOL;
	wNMTInhibitTime : WORD;
	
	udiNumberOfSlaves : UDINT; //How many slaves are attached below the CANopenManager
	udiNumberOfOperationalSlaves : UDINT; //How many slaves are in OPERATIONAL
	udiTotalConfigurationErrors : UDINT; //How many configuration errors (= SDO aborts) happened in configuration phase?
	udiNumberOfSlavesWithActivatedErrorControl : UDINT; //How many slaves have Error control (= Heartbeat or Nodeguarding) activated?
	
	usiCurrentNodeID : USINT;
	
	xEventHandlerRegistered : BOOL;
	EventHandler : CANopenManagerEventHandler; // CANopenManager event handler instance
END_VAR

//gets the CANopenManager kernel state ==> see also CiA405.GET_CANOPEN_KERNEL_STATE
kernelState := CANopen_Manager.KernelState;

//Are all mandatory slaves found and configured by CANopenManager?
xAllMandatorySlaveBooted := CANopen_Manager.MandatorySlavesBooted;

//Are all optional slaves found and configured by CANopenManager?
xAllOptionalSlavesBooted := CANopen_Manager.OptionalSlavesBooted;

//Gets or sets the NMT Inhibit Time (unit: multiple of 100us).
wNMTInhibitTime := CANopen_Manager.NMTInhibitTime;

//go through all remote devices of CANopen_Manager and collect some statistics
udiNumberOfSlaves := 0;
udiNumberOfOperationalSlaves := 0;
udiTotalConfigurationErrors := 0;
udiNumberOfSlavesWithActivatedErrorControl := 0;

FOR usiCurrentNodeID := 1 TO 127 DO
	pDevice := CANopen_Manager.GetSlaveByNodeID(usiCurrentNodeID);
	IF pDevice <> 0 THEN
		//count slaves
		udiNumberOfSlaves := udiNumberOfSlaves + 1;
		
		//Get the slave state ==> see also CiA405.GET_STATE
		IF pDevice^.CANopenState = _3SCOS.DEVICE_STATE.OPERATIONAL THEN
			udiNumberOfOperationalSlaves := udiNumberOfOperationalSlaves + 1;
		END_IF
		
		//Sum up configuration errors. 
		//NOTE: For getting more detailed information you can add the Compiler Define CANOPEN_DEBUG to the application.
		//Then perform a new download and go to the PLC logger. It contains further information for debugging purpose. 
		udiTotalConfigurationErrors := udiTotalConfigurationErrors + pDevice^.ConfigurationErrors;
		
		//Sum up all slaves with error control activated
		IF pDevice^.ErrorControlActivated THEN
			udiNumberOfSlavesWithActivatedErrorControl := udiNumberOfSlavesWithActivatedErrorControl + 1;
		END_IF
	END_IF
END_FOR

// Register a CANopen Manager event handler: An event handler can be used to add additional code to the stack state machine.
// In this example a SDO Read for CANopenRemoteDevice is performed after SDO configuration phase.
// For further details see CANopenManagerEventHandler.EventCallback
IF NOT xEventHandlerRegistered THEN
	xEventHandlerRegistered := CANopen_Manager.RegisterEventHandler(EventHandler);
END_IF

END_PROGRAM

// XC204/Application/CANopen Master Examples/Stack API/Events/CANopenManagerEventHandler
// The following function block shows how to implement a CANopenEventHandler which could be registered
// at CANopen_Manager function block instance (see PRG CANopenManagerAPI).
// See EventCallback method for more details.
FUNCTION_BLOCK CANopenManagerEventHandler IMPLEMENTS _3SCOS.ICANopenEventHandler //Interface needed for registering at CANopen_Manager instance.
VAR_INPUT
END_VAR
VAR_OUTPUT
END_VAR
VAR
	read: CIA405.SDO_READ4; // used to read the device type
	dwDeviceTypeRead : DWORD; // device type read from CANopenRemoteDevice
	xDeviceTypeValid : BOOL; // device type read successfully
END_VAR

// Nothing to do!

// This method implements a CANopen Manager event handler.
// Every time the SDO configuration phase for CANopenRemoteDevice has finished, the Device Type will be read by this handler.
// As long as Event Handler returns FALSE the state machine of CANopenRemoteDevice is stopped. 
METHOD EventCallback : BOOL
VAR_INPUT
	(*Event Type*)
	eEvent	: _3SCOS.CANopenEvent;
	(*NodeID associated with the event; 0 if not relevant.*)
	usiNodeID	: USINT;
END_VAR
CASE eEvent OF
	_3SCOS.CANopenEvent.AFTER_SDO_CONFIG:
		IF usiNodeID = XN_312_GW_CAN.NodeID THEN
			//Read Device Type of slave
			read(ENABLE := TRUE, NETWORK := CANbus.NetId + 1, DEVICE := usiNodeID, CHANNEL := 0, INDEX := 16#1000, SUBINDEX := 16#0);
			IF read.CONFIRM OR read.ERROR <> CIA405.CANOPEN_KERNEL_ERROR.CANOPEN_KERNEL_NO_ERROR THEN
				IF read.CONFIRM THEN
					//value was read without error
					// ==> Copy data from SDO read function block
					MEMUtils.MemCpy(pbyDest := ADR(dwDeviceTypeRead), pbySrc := ADR(read.DATA[1]), dwSize := SIZEOF(dwDeviceTypeRead));
					//==> On big endian systems: dwValue has to be swapped to CANopen byte order (= Little Endian).
					MEMUtils.SwapLocalToIntel(pAddress := ADR(dwDeviceTypeRead), iSize := TO_INT(SIZEOF(dwDeviceTypeRead))); //function only swaps on big endian systems
					xDeviceTypeValid := TRUE;
				ELSE
					xDeviceTypeValid := FALSE;
				END_IF
				
				read(ENABLE := FALSE);
				EventCallback := TRUE; //Event handled ==> resume state machine of CANopenRemoteDevice
			END_IF
		ELSE
			EventCallback := TRUE; // no specific handling for other nodes
		END_IF
	ELSE
		EventCallback := TRUE; // no specific handling for other events
END_CASE
END_METHOD

END_FUNCTION_BLOCK

// XC204/Application/CANopen Master Examples/Stack API/CANopenRemoteDeviceAPI
// This example program shows how to use the CANopen Remotedevice API.
PROGRAM CANopenRemoteDeviceAPI
VAR
	slaveState : _3SCOS.DEVICE_STATE;
	uiConfigurationErrors : UINT;
	xErrorControlActivated : BOOL;
	pCANopenManager : POINTER TO _3SCOS.CANopenManager;
END_VAR

//Gets the pointer to the CANopenManager
pCANopenManager := XN_312_GW_CAN.pCANopenManager;

//Set Bootup Timeout of slave to 10 seconds
XN_312_GW_CAN.BootupTimeout := 10000000; // unit: us
		
//Get the slave state ==> see also CiA405.GET_STATE
slaveState := XN_312_GW_CAN.CANopenState;

//How many configuration errors (= SDO aborts) happened in configuration phase of the slave?
uiConfigurationErrors := XN_312_GW_CAN.ConfigurationErrors;

//Error control (= Heartbeat or Nodeguarding) for slave activated?
xErrorControlActivated := XN_312_GW_CAN.ErrorControlActivated;

//Set the NMT Error behaviour of slave to RESTART_SLAVE.
//This means: If a Heartbeat or Nodeguarding error is detected for the slave it will be automatically restarted (=default behaviour).
XN_312_GW_CAN.NMTErrorBehaviour := _3SCOS.NMT_ERROR_BEHAVIOUR.RESTART_SLAVE;

END_PROGRAM

// XC204/Application/CANbus Examples/CANbusExamples
PROGRAM CANbusExamples
VAR
END_VAR

ChangeBaudrate(); // How to change the baudrate of a CANbus
EnableDisableCANbus(); // How to enable/disable a CANbus

END_PROGRAM

// XC204/Application/CANbus Examples/Change CANbus settings (Reconfigure)/ChangeBaudrate
// This program shows how to change the baudrate of a CANbus by using CAA Device Diagnosis Reconfigure.
// Make sure that PLC setting "Enable Diagnosis for devices" is activated!
// Set xEnable to TRUE in online mode to get the program working.
PROGRAM ChangeBaudrate
VAR
	xEnable       : BOOL; // Set this variable to true to start the example code.
	usiNetID	  : USINT; // NetID of CANbus on which baudrate change should be performed
	wBaudrate : WORD := 1000; // Set new Baudrate 
	
	iState : INT := 0;
	pCANBus : POINTER TO CANbusDevice.CANbus_Diag;
	reconfigure : DED.Reconfigure;
	RTrig 	 : Standard.R_TRIG;
END_VAR

CASE iState OF
	0:
		//Detect rising edge
		RTrig(CLK := xEnable);
		IF RTrig.Q THEN
			iState := 1;
		END_IF	

	1: 
		// Get the CANbus instance for a specific Network ID
		pCANBus := GetCANbus(usiNetID); // Here the pointer to the CANbus instance with NetID = usiNetID is calculated (the generic way!), 
									    // but you can also use the CANbus FB instance directly. For example: CANbus_1.SetBaudrate(wBaudrate)
		IF pCANBus <> 0 THEN
			// CANbus found ==> Set new Baudrate. Note: Baudrate change takes effect after reconfigure.
			// It is also possible changing NetID by calling SetNetID.
			pCANBus^.SetBaudrate(wBaudrate);
			iState := 2;
		ELSE
			// Error : No CANbus found
			iState := 3;
		END_IF
		
	2:
		// perform reconfigure
		reconfigure(xExecute := TRUE, itfNode := pCANBus^); // Here we use the pointer to the CANbus and dereference it. 
															// So we get the INode interface which is implemented by this instance (==> the generic way). 
															// But you can also use the CANbus FB instance directly. For Example: reconfigure(xExecute := TRUE, itfNode := CANbus_1)
		
		IF reconfigure.xDone OR reconfigure.xError THEN 	// Note: Add error handling for xError!
			reconfigure(xExecute := FALSE);
			iState := 3;
		END_IF
		
	3:
		iState := 0;
		xEnable := FALSE;
END_CASE

END_PROGRAM

// XC204/Application/CANbus Examples/Query CANbus/GetCANbus
// Gets the pointer to the CANbus device instance by using CAA Device Diagnosis and __QUERYPOINTER.
// Make sure that PLC setting "Enable Diagnosis for devices" is activated!
FUNCTION GetCANbus : POINTER TO CANbusDevice.CANbus_Diag
VAR_INPUT
	usiNetID : USINT; // Network ID of CANbus
END_VAR
VAR
	itfNode : DED.INode;
	itfBus : DED.IBus;
	buiBusInfo : DED.BUS_INFO;
END_VAR

// first get PLC device
itfNode := DED.GetRoot();

// Go through device tree and search for CANbus
WHILE itfNode <> 0 DO
	itfBus := DED.INode_TO_IBus(itfNode); // check if current node is a bus
	IF itfBus <> 0 THEN
		// current node is a bus
		IF itfBus.GetBusInfo(buiBusInfo) = DED.ERROR.NO_ERROR THEN // get bus information
			IF buiBusInfo.eType = DED.BUS_TYPE.CAN AND_THEN buiBusInfo.idSystem = usiNetID THEN //check if it is a CANbus and compare NetID
				// CANbus found!
				__QUERYPOINTER(itfBus, GetCANbus); // Get CANbus_Diag instance pointer
				EXIT; // finished!
			END_IF
		END_IF
	END_IF
	
	itfBus := 0;
	itfNode := DED.GetNextNode(itfNode); // traverse tree ==> go to next node
END_WHILE

END_FUNCTION

// XC204/Application/CANbus Examples/Change CANbus settings (Reconfigure)/EnableDisableCANbus
// This program shows how to enable/disable a complete CANbus by using CAA Device Diagnosis Reconfigure.
// This example project is not only appliable on CANbus nodes. It works also on all other nodes (e.g. CANopen Manager, CANopen Local Device, ...).
// Make sure that PLC setting "Enable Diagnosis for devices" is activated!
// Set xEnable to TRUE in online mode to get the program working.
PROGRAM EnableDisableCANbus
VAR
	xEnable       : BOOL; // Set this variable to true to start the example code.
	usiNetID	  : USINT; // NetID of CANbus which should be enabled/disabled
	xEnableCANbus : BOOL; // TRUE: Enable CANbus, FALSE: Disable CANbus
	
	iState : INT := 0;
	
	pCANbus : POINTER TO CANbusDevice.CANbus_Diag;
	reconfigure : DED.Reconfigure;
	RTrig 	 : Standard.R_TRIG;
END_VAR

CASE iState OF
	0:
		//Detect rising edge
		RTrig(CLK := xEnable);
		IF RTrig.Q THEN
			iState := 1;
		END_IF
	1:
		// Get the CANbus instance for a specific Network ID
		pCANbus := GetCANbus(usiNetID);
		
		IF pCANbus <> 0 THEN
			// CANbus found ==> Set enable flag. Note: Enable flag takes effect after reconfigure.
			pCANbus^.Enable := xEnableCANbus;
			iState := 2;
		ELSE
			// Error : No CANbus found
			iState := 3;
		END_IF
		
	2:
		// perform reconfigure
		reconfigure(xExecute := TRUE, itfNode := pCANbus^); // Here we use the pointer to the CANbus and dereference it.
															// So we get the INode interface which is implemented by this instance (==> the generic way). 
															// But you can also use the CANbus FB instance directly. For Example: reconfigure(xExecute := TRUE, itfNode := CANbus_1)

		IF reconfigure.xDone OR reconfigure.xError THEN     // Note: Add error handling for xError!
			reconfigure(xExecute := FALSE);
			iState := 3;
		END_IF
		
	3:
		iState := 0;
		xEnable := FALSE;
END_CASE

END_PROGRAM
